// TIA Portal project "14_Palletizer_System" (V19)

(* hardware
DEVICE "S7-1500/ET200MP station_1"  S7-1500 station
   slot 0: "Rail_0"  Rack  6ES7 590-1***0-0AA0
   slot 1: "PLC_1"  CPU 1513-1 PN  6ES7 513-1AL02-0AB0  V2.9
      slot 3: "CPU display_1"  6ES7591-1AA00-0AA0
      slot 32768: "PROFINET interface_1"  X1
         slot 32769: "Port_1"  X1 P1
         slot 32770: "Port_2"  X1 P2
      slot 34817: "Virtual CP interface port_1"  Virtual CP interface port  Virtual CP interface port
*)

// ===== PLC "PLC_1"  CPU 1513-1 PN =====

VAR_GLOBAL   // PLC tag table "Default tag table"
   "Start" AT %I0.0 : Bool;
   "Stop" AT %I0.1 : Bool;
   "Reset" AT %I0.2 : Bool;
   "Auto" AT %I0.3 : Bool;
   "Manual" AT %I0.4 : Bool;
   "Box at entry" AT %I0.5 : Bool;
   "Clamped" AT %I0.6 : Bool;
   "Elevator moving" AT %I0.7 : Bool;
   "Pallet at entry" AT %I1.0 : Bool;
   "Pallet at exit" AT %I1.1 : Bool;
   "Pallet loaded" AT %I1.2 : Bool;
   "Plate limit" AT %I1.3 : Bool;
   "Pusher limit" AT %I1.4 : Bool;
   "Start light" AT %Q0.0 : Bool;
   "Stop light" AT %Q0.1 : Bool;
   "Reset light" AT %Q0.2 : Bool;
   "Clamp" AT %Q0.3 : Bool;
   "Box feeder" AT %Q0.4 : Bool;
   "Elevator up" AT %Q0.5 : Bool;
   "Elevator down" AT %Q0.6 : Bool;
   "Exit conveyor" AT %Q0.7 : Bool;
   "Load belt" AT %Q1.0 : Bool;
   "Load pallet" AT %Q1.1 : Bool;
   "Move to limit" AT %Q1.2 : Bool;
   "Open plate" AT %Q1.3 : Bool;
   "Pallet feeder" AT %Q1.4 : Bool;
   "Push" AT %Q1.5 : Bool;
   "Turn" AT %Q1.6 : Bool;
   "Warning light" AT %Q1.7 : Bool;
   "Set the value for the set of boxes" AT %ID30 : Real;
   "Counter" AT %QD30 : DInt;
   "Display for the set of box" AT %QD34 : DInt;
   "nw2" AT %M0.0 : Bool;
   "nw3 2nd memory" AT %M0.2 : Bool;
   "nw3 1st memory (Unpause)" AT %M0.1 : Bool;
   "nw4 pl p" AT %M1.1 : Bool;
   "nw4" AT %M0.3 : Bool;
   "nw4 op n" AT %M3.6 : Bool;
   "nw4 bae p" AT %M1.4 : Bool;
   "nw5" AT %M0.4 : Bool;
   "nw5 pl p" AT %M1.0 : Bool;
   "nw5 op n" AT %M3.7 : Bool;
   "nw6 bae n" AT %M1.2 : Bool;
   "nw6 bae p" AT %M1.3 : Bool;
   "nw6" AT %M4.0 : Bool;
   "nw6 pl p reset DB1" AT %M0.7 : Bool;
   "nw6 pl p" AT %M4.1 : Bool;
   "nw7 pae p" AT %M5.7 : Bool;
   "nw7" AT %M1.6 : Bool;
   "nw7 pl p" AT %M6.3 : Bool;
   "nw8 pae n" AT %M6.4 : Bool;
   "O/P for DB4 nw15" AT %M5.4 : Bool;
   "nw8" AT %M1.7 : Bool;
   "nw8 em n" AT %M6.0 : Bool;
   "nw8 pl p" AT %M2.6 : Bool;
   "nw9 pl p" AT %M2.4 : Bool;
   "nw9" AT %M2.0 : Bool;
   "nw9 em n" AT %M2.2 : Bool;
   "nw10 pl p" AT %M6.2 : Bool;
   "nw10" AT %M2.1 : Bool;
   "nw10 em n" AT %M2.3 : Bool;
   "nw10 pae p" AT %M6.1 : Bool;
   "nw11 p n" AT %M2.5 : Bool;
   "nw11" AT %M4.5 : Bool;
   "nw11 ed p reset CTU" AT %M3.5 : Bool;
   "nw11 ed p reset SR" AT %M4.6 : Bool;
   "nw13 pl p" AT %M3.1 : Bool;
   "nw13" AT %M3.4 : Bool;
   "nw12 c n" AT %M3.0 : Bool;
   "nw12" AT %M2.7 : Bool;
   "nw12 em n" AT %M3.2 : Bool;
   "nw13 pae p" AT %M5.6 : Bool;
   "nw14 p n" AT %M0.5 : Bool;
   "nw14 op n" AT %M4.4 : Bool;
   "nw14" AT %M4.2 : Bool;
   "nw14 ed p reset CTU" AT %M0.6 : Bool;
   "nw14 c n reset SR" AT %M4.3 : Bool;
   "nw15 ed n" AT %M4.7 : Bool;
   "nw15 pae p" AT %M5.0 : Bool;
   "Set the value for boxes on the display" AT %MW100 : Int;
   "nw16 pae n" AT %M5.1 : Bool;
   "nw16" AT %M5.3 : Bool;
   "nw16 eu p" AT %M6.7 : Bool;
   "nw17 bae n" AT %M6.5 : Bool;
   "nw18" AT %M6.6 : Bool;
   "nw13 op n" AT %M3.3 : Bool;
END_VAR

// folder: System blocks/Program resources

DATA_BLOCK "IEC_Counter_0_DB"   // DB1
{ S7_Optimized_Access := 'TRUE' }
AUTHOR : Simatic
FAMILY : IEC
NAME : CNTR
VERSION : 1.0
// stored: InstanceOfName IEC_COUNTER
"IEC_COUNTER"
BEGIN
END_DATA_BLOCK

DATA_BLOCK "IEC_Counter_0_DB_1"   // DB2
{ S7_Optimized_Access := 'TRUE' }
AUTHOR : Simatic
FAMILY : IEC
NAME : CNTR
VERSION : 1.0
// stored: InstanceOfName IEC_COUNTER
"IEC_COUNTER"
BEGIN
END_DATA_BLOCK

DATA_BLOCK "CTU to turn the box"   // DB3
{ S7_Optimized_Access := 'TRUE' }
AUTHOR : Simatic
FAMILY : IEC
NAME : CNTR
VERSION : 1.0
// stored: InstanceOfName IEC_COUNTER
"IEC_COUNTER"
BEGIN
END_DATA_BLOCK

DATA_BLOCK "Count a set of boxes that are moved on the pallet"   // DB4
{ S7_Optimized_Access := 'TRUE' }
AUTHOR : Simatic
FAMILY : IEC
NAME : CNTR
VERSION : 1.0
// stored: InstanceOfName IEC_COUNTER
"IEC_COUNTER"
BEGIN
END_DATA_BLOCK

DATA_BLOCK "Count total number of boxes that are moved on the pallet"   // DB5
{ S7_Optimized_Access := 'TRUE' }
AUTHOR : Simatic
FAMILY : IEC
NAME : CNTR
VERSION : 1.0
// stored: InstanceOfName IEC_COUNTER
"IEC_COUNTER"
BEGIN
END_DATA_BLOCK

// folder: (top level)

ORGANIZATION_BLOCK "Main"   // OB1, LAD, ProgramCycle
TITLE = "Main Program Sweep (Cycle)"
{ S7_Optimized_Access := 'TRUE' }
VERSION : 0.1
   VAR_INPUT
      Initial_Call : Bool;   // Initial call of this OB
      Remanence : Bool;   // =True, if remanent data are available
   END_VAR
   VAR_TEMP   // added for the SCL form of the ladder/FBD networks
      _w1 : Bool;
      _w2 : Bool;
      _w3 : Bool;
      _w4 : Bool;
   END_VAR
BEGIN

REGION Network 2: Start or Reset System with LED ON/OFF which are mounted on the switches
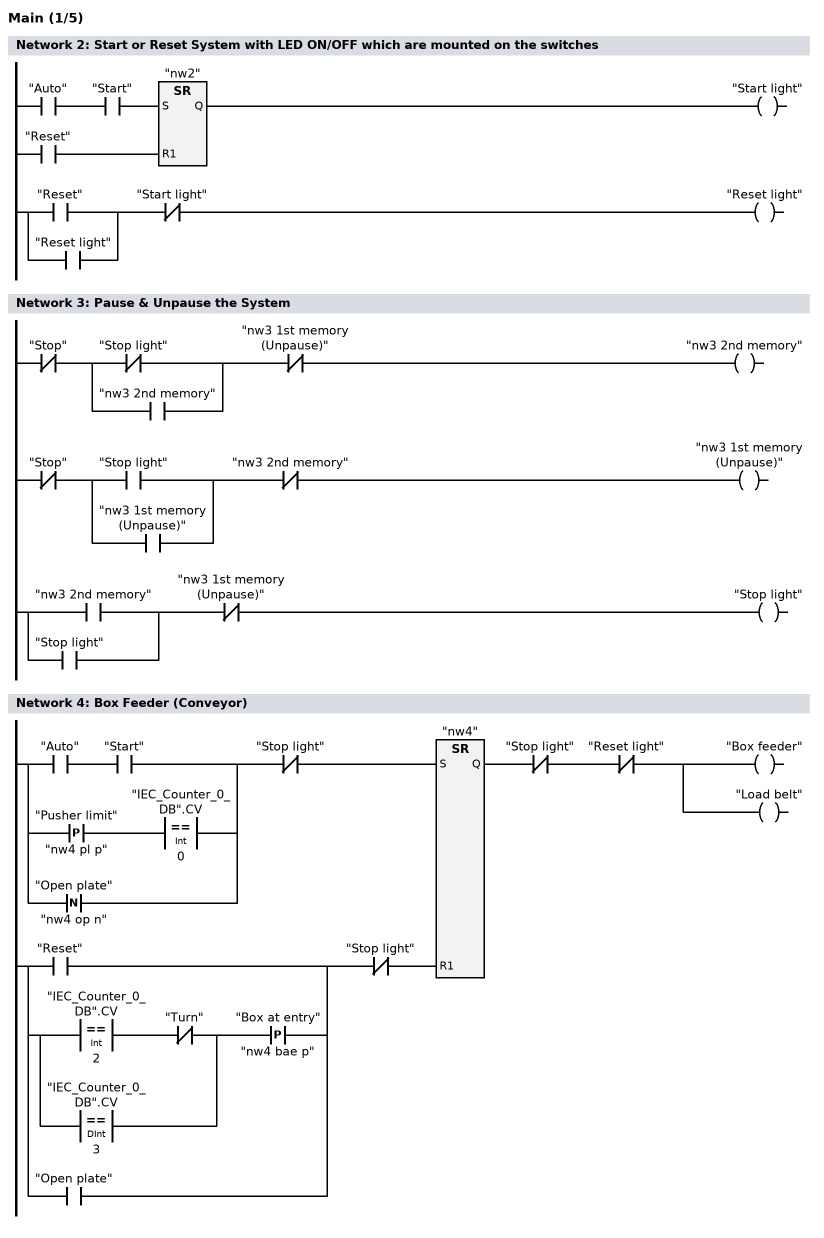
   RUNG wire#powerrail
      Contact( "Auto" )
      Contact( "Start" )
      S_SR(operand := "nw2", r1 := wire#w1)
      Coil( "Start light" )
   END_RUNG
   RUNG wire#powerrail
      Contact( "Reset" )
   END_RUNG wire#w1
   RUNG wire#powerrail
      Contact( "Reset" )
      wire#w2
      I_Contact( "Start light" )
      Coil( "Reset light" )
   END_RUNG
   RUNG wire#powerrail
      Contact( "Reset light" )
   END_RUNG wire#w2
   // the same network as SCL:
   IF "Auto" AND "Start" THEN
       "nw2" := TRUE;   // SR flip-flop
   END_IF;
   IF "Reset" THEN "nw2" := FALSE; END_IF;
   "Start light" := "nw2";
   "Reset light" := ("Reset" OR "Reset light") AND NOT "Start light";
END_REGION

REGION Network 3: Pause & Unpause the System
   RUNG wire#powerrail
      I_Contact( "Stop" )
      wire#w1
      I_Contact( "Stop light" )
      wire#w2
      I_Contact( "nw3 1st memory (Unpause)" )
      Coil( "nw3 2nd memory" )
   END_RUNG
   RUNG wire#w1
      Contact( "nw3 2nd memory" )
   END_RUNG wire#w2
   RUNG wire#powerrail
      I_Contact( "Stop" )
      wire#w3
      Contact( "Stop light" )
      wire#w4
      I_Contact( "nw3 2nd memory" )
      Coil( "nw3 1st memory (Unpause)" )
   END_RUNG
   RUNG wire#w3
      Contact( "nw3 1st memory (Unpause)" )
   END_RUNG wire#w4
   RUNG wire#powerrail
      Contact( "nw3 2nd memory" )
      wire#w5
      I_Contact( "nw3 1st memory (Unpause)" )
      Coil( "Stop light" )
   END_RUNG
   RUNG wire#powerrail
      Contact( "Stop light" )
   END_RUNG wire#w5
   // the same network as SCL:
   "nw3 2nd memory" := NOT "Stop" AND (NOT "Stop light" OR "nw3 2nd memory") AND NOT "nw3 1st memory (Unpause)";
   "nw3 1st memory (Unpause)" := NOT "Stop" AND ("Stop light" OR "nw3 1st memory (Unpause)") AND NOT "nw3 2nd memory";
   "Stop light" := ("nw3 2nd memory" OR "Stop light") AND NOT "nw3 1st memory (Unpause)";
END_REGION

REGION Network 4: Box Feeder (Conveyor)
   RUNG wire#powerrail
      Contact( "Auto" )
      Contact( "Start" )
      wire#w1
      I_Contact( "Stop light" )
      S_SR(operand := "nw4", r1 := wire#w4)
      I_Contact( "Stop light" )
      I_Contact( "Reset light" )
      wire#w5
      Coil( "Box feeder" )
   END_RUNG
   RUNG wire#powerrail
      P_Contact(operand := "Pusher limit", bit := "nw4 pl p")
      { S7_Templates := "SrcType := Int" } EQ_Contact(in1 := "IEC_Counter_0_DB".CV, in2 := 0)
   END_RUNG wire#w1
   RUNG wire#powerrail
      N_Contact(operand := "Open plate", bit := "nw4 op n")
   END_RUNG wire#w1
   RUNG wire#powerrail
      Contact( "Reset" )
      wire#w2
      I_Contact( "Stop light" )
   END_RUNG wire#w4
   RUNG wire#powerrail
      { S7_Templates := "SrcType := Int" } EQ_Contact(in1 := "IEC_Counter_0_DB".CV, in2 := 2)
      I_Contact( "Turn" )
      wire#w3
      P_Contact(operand := "Box at entry", bit := "nw4 bae p")
   END_RUNG wire#w2
   RUNG wire#powerrail
      { S7_Templates := "SrcType := DInt" } EQ_Contact(in1 := "IEC_Counter_0_DB".CV, in2 := 3)
   END_RUNG wire#w3
   RUNG wire#powerrail
      Contact( "Open plate" )
   END_RUNG wire#w2
   RUNG wire#w5
      Coil( "Load belt" )
   END_RUNG
   // the same network as SCL:
   #_w1 := "Pusher limit" AND NOT "nw4 pl p";   // rising edge of "Pusher limit"
   "nw4 pl p" := "Pusher limit";
   #_w2 := NOT "Open plate" AND "nw4 op n";   // falling edge of "Open plate"
   "nw4 op n" := "Open plate";
   #_w3 := ((("IEC_Counter_0_DB".CV = 2) AND NOT "Turn") OR ("IEC_Counter_0_DB".CV = 3)) AND "Box at entry" AND NOT "nw4 bae p";   // rising edge of "Box at entry"
   "nw4 bae p" := "Box at entry";
   IF (("Auto" AND "Start") OR (#_w1 AND ("IEC_Counter_0_DB".CV = 0)) OR #_w2) AND NOT "Stop light" THEN
       "nw4" := TRUE;   // SR flip-flop
   END_IF;
   IF ("Reset" OR #_w3 OR "Open plate") AND NOT "Stop light" THEN "nw4" := FALSE; END_IF;
   "Box feeder" := "nw4" AND NOT "Stop light" AND NOT "Reset light";
   "Load belt" := "Box feeder";
END_REGION

REGION Network 5: Load Belt Conveyor (Move to Network 4 for Optimizer)
END_REGION

REGION Network 6: Push and Push Limit
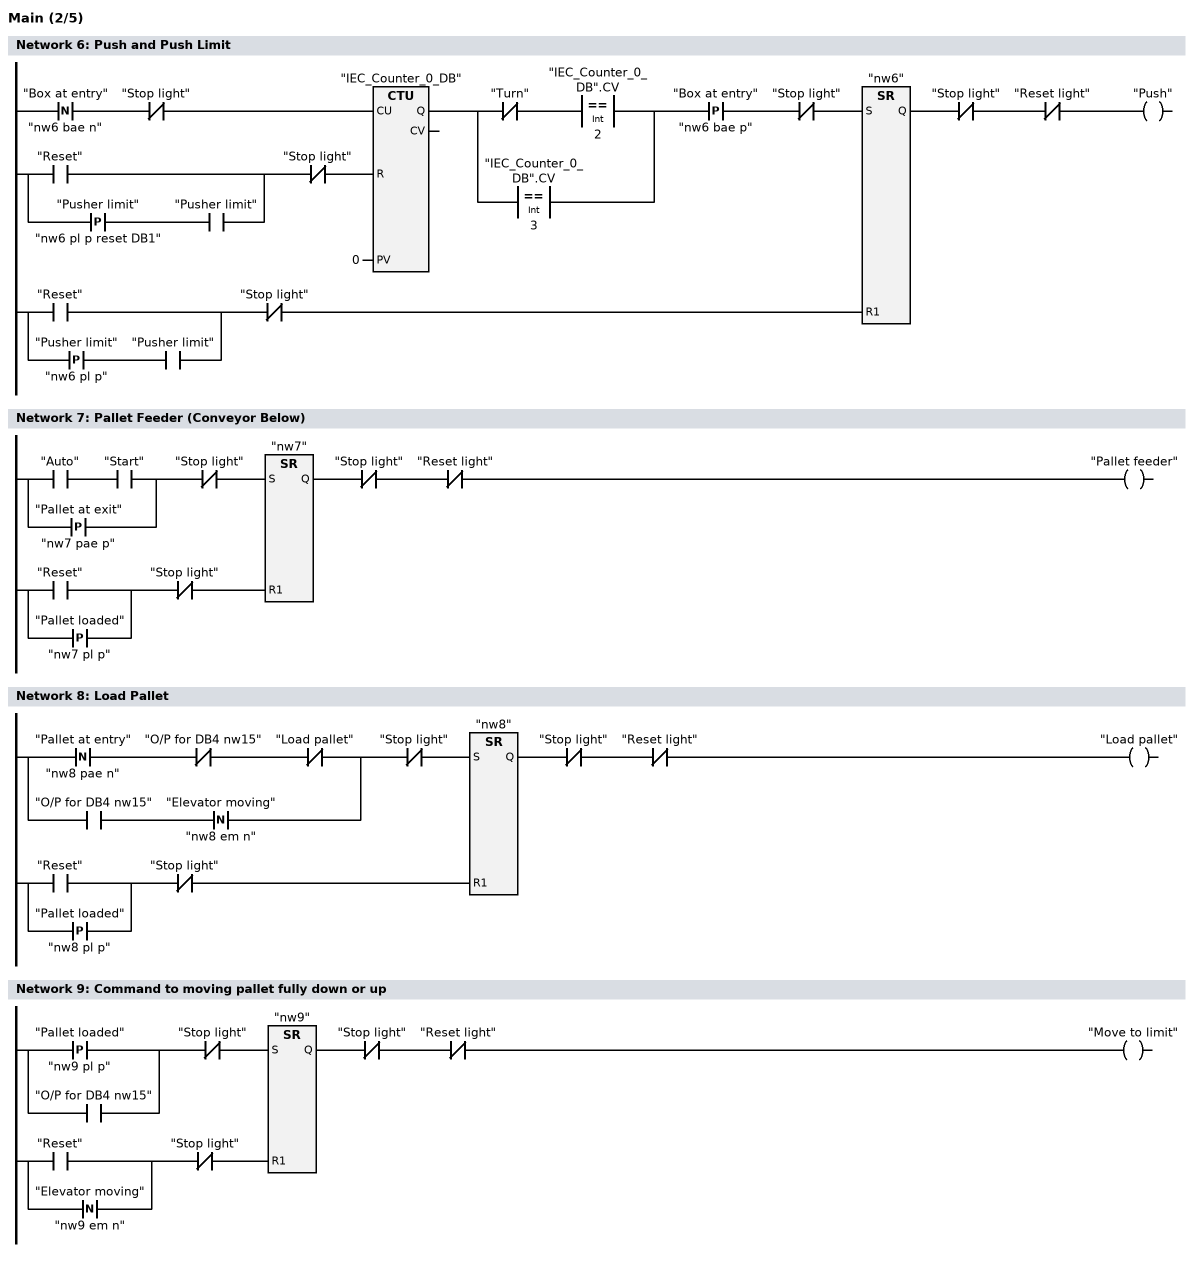
   #_w1 := NOT "Box at entry" AND "nw6 bae n";   // falling edge of "Box at entry"
   "nw6 bae n" := "Box at entry";
   #_w2 := "Pusher limit" AND NOT "nw6 pl p reset DB1";   // rising edge of "Pusher limit"
   "nw6 pl p reset DB1" := "Pusher limit";
   "IEC_Counter_0_DB".CTU(CU := #_w1 AND NOT "Stop light",
                          R := ("Reset" OR (#_w2 AND "Pusher limit")) AND NOT "Stop light",
                          PV := 0);
   #_w3 := "IEC_Counter_0_DB".Q AND ((NOT "Turn" AND ("IEC_Counter_0_DB".CV = 2)) OR ("IEC_Counter_0_DB".CV = 3)) AND "Box at entry" AND NOT "nw6 bae p";   // rising edge of "Box at entry"
   "nw6 bae p" := "Box at entry";
   #_w4 := "Pusher limit" AND NOT "nw6 pl p";   // rising edge of "Pusher limit"
   "nw6 pl p" := "Pusher limit";
   IF #_w3 AND NOT "Stop light" THEN
       "nw6" := TRUE;   // SR flip-flop
   END_IF;
   IF ("Reset" OR (#_w4 AND "Pusher limit")) AND NOT "Stop light" THEN "nw6" := FALSE; END_IF;
   "Push" := "nw6" AND NOT "Stop light" AND NOT "Reset light";
END_REGION

REGION Network 7: Pallet Feeder (Conveyor Below)
   RUNG wire#powerrail
      Contact( "Auto" )
      Contact( "Start" )
      wire#w1
      I_Contact( "Stop light" )
      S_SR(operand := "nw7", r1 := wire#w3)
      I_Contact( "Stop light" )
      I_Contact( "Reset light" )
      Coil( "Pallet feeder" )
   END_RUNG
   RUNG wire#powerrail
      P_Contact(operand := "Pallet at exit", bit := "nw7 pae p")
   END_RUNG wire#w1
   RUNG wire#powerrail
      Contact( "Reset" )
      wire#w2
      I_Contact( "Stop light" )
   END_RUNG wire#w3
   RUNG wire#powerrail
      P_Contact(operand := "Pallet loaded", bit := "nw7 pl p")
   END_RUNG wire#w2
   // the same network as SCL:
   #_w1 := "Pallet at exit" AND NOT "nw7 pae p";   // rising edge of "Pallet at exit"
   "nw7 pae p" := "Pallet at exit";
   #_w2 := "Pallet loaded" AND NOT "nw7 pl p";   // rising edge of "Pallet loaded"
   "nw7 pl p" := "Pallet loaded";
   IF (("Auto" AND "Start") OR #_w1) AND NOT "Stop light" THEN
       "nw7" := TRUE;   // SR flip-flop
   END_IF;
   IF ("Reset" OR #_w2) AND NOT "Stop light" THEN "nw7" := FALSE; END_IF;
   "Pallet feeder" := "nw7" AND NOT "Stop light" AND NOT "Reset light";
END_REGION

REGION Network 8: Load Pallet
   RUNG wire#powerrail
      N_Contact(operand := "Pallet at entry", bit := "nw8 pae n")
      I_Contact( "O/P for DB4 nw15" )
      I_Contact( "Load pallet" )
      wire#w1
      I_Contact( "Stop light" )
      S_SR(operand := "nw8", r1 := wire#w3)
      I_Contact( "Stop light" )
      I_Contact( "Reset light" )
      Coil( "Load pallet" )
   END_RUNG
   RUNG wire#powerrail
      Contact( "O/P for DB4 nw15" )
      N_Contact(operand := "Elevator moving", bit := "nw8 em n")
   END_RUNG wire#w1
   RUNG wire#powerrail
      Contact( "Reset" )
      wire#w2
      I_Contact( "Stop light" )
   END_RUNG wire#w3
   RUNG wire#powerrail
      P_Contact(operand := "Pallet loaded", bit := "nw8 pl p")
   END_RUNG wire#w2
   // the same network as SCL:
   #_w1 := NOT "Pallet at entry" AND "nw8 pae n";   // falling edge of "Pallet at entry"
   "nw8 pae n" := "Pallet at entry";
   #_w2 := "O/P for DB4 nw15" AND NOT "Elevator moving" AND "nw8 em n";   // falling edge of "Elevator moving"
   "nw8 em n" := "Elevator moving";
   #_w3 := "Pallet loaded" AND NOT "nw8 pl p";   // rising edge of "Pallet loaded"
   "nw8 pl p" := "Pallet loaded";
   IF ((#_w1 AND NOT "O/P for DB4 nw15" AND NOT "Load pallet") OR #_w2) AND NOT "Stop light" THEN
       "nw8" := TRUE;   // SR flip-flop
   END_IF;
   IF ("Reset" OR #_w3) AND NOT "Stop light" THEN "nw8" := FALSE; END_IF;
   "Load pallet" := "nw8" AND NOT "Stop light" AND NOT "Reset light";
END_REGION

REGION Network 9: Command to moving pallet fully down or up
   RUNG wire#powerrail
      P_Contact(operand := "Pallet loaded", bit := "nw9 pl p")
      wire#w1
      I_Contact( "Stop light" )
      S_SR(operand := "nw9", r1 := wire#w3)
      I_Contact( "Stop light" )
      I_Contact( "Reset light" )
      Coil( "Move to limit" )
   END_RUNG
   RUNG wire#powerrail
      Contact( "O/P for DB4 nw15" )
   END_RUNG wire#w1
   RUNG wire#powerrail
      Contact( "Reset" )
      wire#w2
      I_Contact( "Stop light" )
   END_RUNG wire#w3
   RUNG wire#powerrail
      N_Contact(operand := "Elevator moving", bit := "nw9 em n")
   END_RUNG wire#w2
   // the same network as SCL:
   #_w1 := "Pallet loaded" AND NOT "nw9 pl p";   // rising edge of "Pallet loaded"
   "nw9 pl p" := "Pallet loaded";
   #_w2 := NOT "Elevator moving" AND "nw9 em n";   // falling edge of "Elevator moving"
   "nw9 em n" := "Elevator moving";
   IF (#_w1 OR "O/P for DB4 nw15") AND NOT "Stop light" THEN
       "nw9" := TRUE;   // SR flip-flop
   END_IF;
   IF ("Reset" OR #_w2) AND NOT "Stop light" THEN "nw9" := FALSE; END_IF;
   "Move to limit" := "nw9" AND NOT "Stop light" AND NOT "Reset light";
END_REGION

REGION Network 10: Move Pallet upward by 1 step or fully up
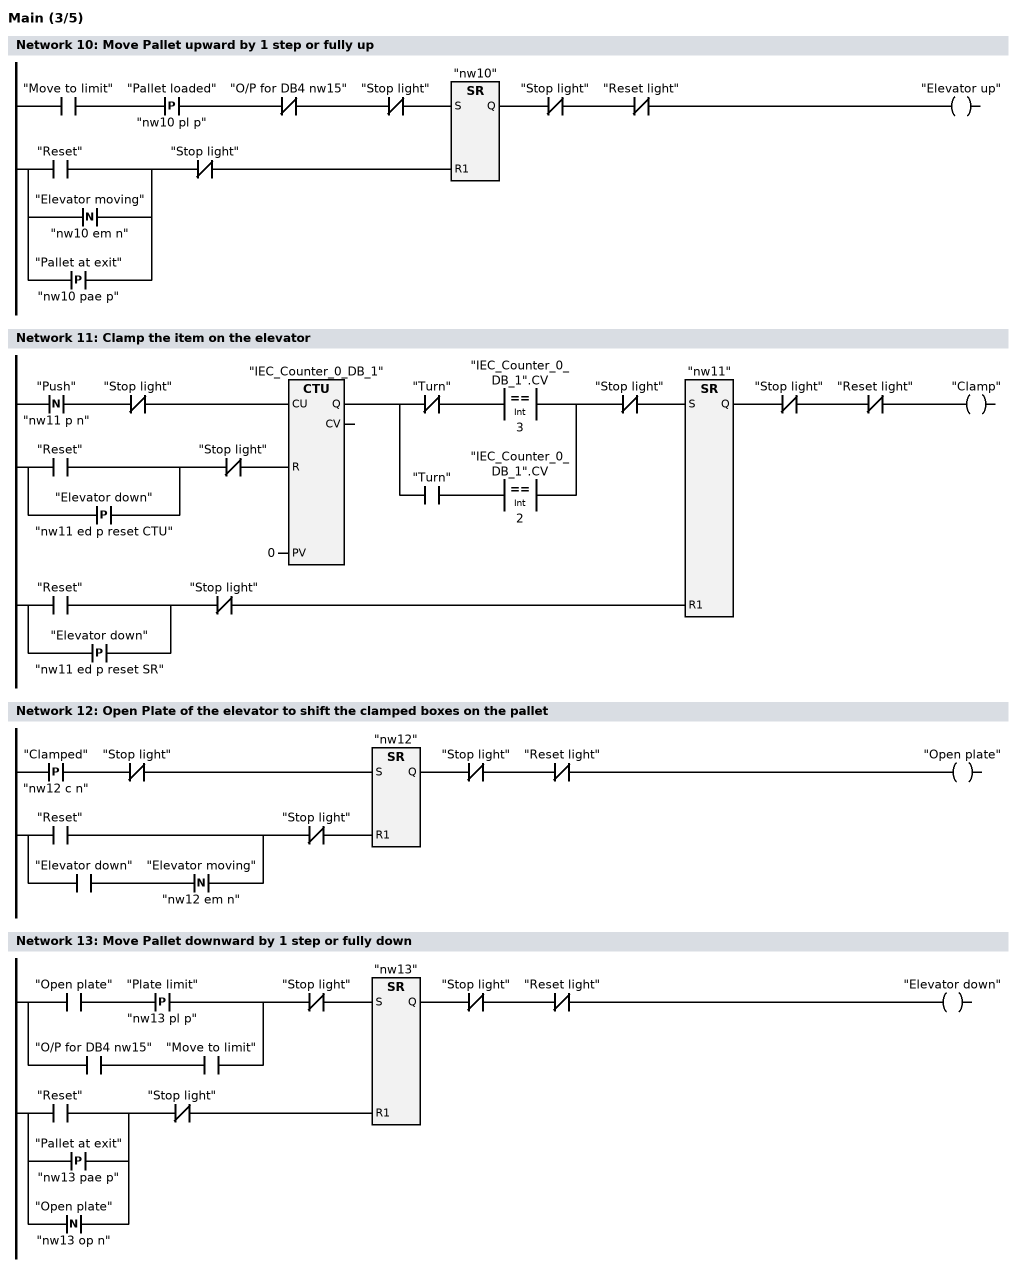
   RUNG wire#powerrail
      Contact( "Move to limit" )
      P_Contact(operand := "Pallet loaded", bit := "nw10 pl p")
      I_Contact( "O/P for DB4 nw15" )
      I_Contact( "Stop light" )
      S_SR(operand := "nw10", r1 := wire#w2)
      I_Contact( "Stop light" )
      I_Contact( "Reset light" )
      Coil( "Elevator up" )
   END_RUNG
   RUNG wire#powerrail
      Contact( "Reset" )
      wire#w1
      I_Contact( "Stop light" )
   END_RUNG wire#w2
   RUNG wire#powerrail
      N_Contact(operand := "Elevator moving", bit := "nw10 em n")
   END_RUNG wire#w1
   RUNG wire#powerrail
      P_Contact(operand := "Pallet at exit", bit := "nw10 pae p")
   END_RUNG wire#w1
   // the same network as SCL:
   #_w1 := "Move to limit" AND "Pallet loaded" AND NOT "nw10 pl p";   // rising edge of "Pallet loaded"
   "nw10 pl p" := "Pallet loaded";
   #_w2 := NOT "Elevator moving" AND "nw10 em n";   // falling edge of "Elevator moving"
   "nw10 em n" := "Elevator moving";
   #_w3 := "Pallet at exit" AND NOT "nw10 pae p";   // rising edge of "Pallet at exit"
   "nw10 pae p" := "Pallet at exit";
   IF #_w1 AND NOT "O/P for DB4 nw15" AND NOT "Stop light" THEN
       "nw10" := TRUE;   // SR flip-flop
   END_IF;
   IF ("Reset" OR #_w2 OR #_w3) AND NOT "Stop light" THEN "nw10" := FALSE; END_IF;
   "Elevator up" := "nw10" AND NOT "Stop light" AND NOT "Reset light";
END_REGION

REGION Network 11: Clamp the item on the elevator
   #_w1 := NOT "Push" AND "nw11 p n";   // falling edge of "Push"
   "nw11 p n" := "Push";
   #_w2 := "Elevator down" AND NOT "nw11 ed p reset CTU";   // rising edge of "Elevator down"
   "nw11 ed p reset CTU" := "Elevator down";
   "IEC_Counter_0_DB_1".CTU(CU := #_w1 AND NOT "Stop light",
                           R := ("Reset" OR #_w2) AND NOT "Stop light",
                           PV := 0);
   #_w3 := "Elevator down" AND NOT "nw11 ed p reset SR";   // rising edge of "Elevator down"
   "nw11 ed p reset SR" := "Elevator down";
   IF "IEC_Counter_0_DB_1".Q AND ((NOT "Turn" AND ("IEC_Counter_0_DB_1".CV = 3)) OR ("Turn" AND ("IEC_Counter_0_DB_1".CV = 2))) AND NOT "Stop light" THEN
       "nw11" := TRUE;   // SR flip-flop
   END_IF;
   IF ("Reset" OR #_w3) AND NOT "Stop light" THEN "nw11" := FALSE; END_IF;
   "Clamp" := "nw11" AND NOT "Stop light" AND NOT "Reset light";
END_REGION

REGION Network 12: Open Plate of the elevator to shift the clamped boxes on the pallet
   RUNG wire#powerrail
      P_Contact(operand := "Clamped", bit := "nw12 c n")
      I_Contact( "Stop light" )
      S_SR(operand := "nw12", r1 := wire#w2)
      I_Contact( "Stop light" )
      I_Contact( "Reset light" )
      Coil( "Open plate" )
   END_RUNG
   RUNG wire#powerrail
      Contact( "Reset" )
      wire#w1
      I_Contact( "Stop light" )
   END_RUNG wire#w2
   RUNG wire#powerrail
      Contact( "Elevator down" )
      N_Contact(operand := "Elevator moving", bit := "nw12 em n")
   END_RUNG wire#w1
   // the same network as SCL:
   #_w1 := "Clamped" AND NOT "nw12 c n";   // rising edge of "Clamped"
   "nw12 c n" := "Clamped";
   #_w2 := "Elevator down" AND NOT "Elevator moving" AND "nw12 em n";   // falling edge of "Elevator moving"
   "nw12 em n" := "Elevator moving";
   IF #_w1 AND NOT "Stop light" THEN
       "nw12" := TRUE;   // SR flip-flop
   END_IF;
   IF ("Reset" OR #_w2) AND NOT "Stop light" THEN "nw12" := FALSE; END_IF;
   "Open plate" := "nw12" AND NOT "Stop light" AND NOT "Reset light";
END_REGION

REGION Network 13: Move Pallet downward by 1 step or fully down
   RUNG wire#powerrail
      Contact( "Open plate" )
      P_Contact(operand := "Plate limit", bit := "nw13 pl p")
      wire#w1
      I_Contact( "Stop light" )
      S_SR(operand := "nw13", r1 := wire#w3)
      I_Contact( "Stop light" )
      I_Contact( "Reset light" )
      Coil( "Elevator down" )
   END_RUNG
   RUNG wire#powerrail
      Contact( "O/P for DB4 nw15" )
      Contact( "Move to limit" )
   END_RUNG wire#w1
   RUNG wire#powerrail
      Contact( "Reset" )
      wire#w2
      I_Contact( "Stop light" )
   END_RUNG wire#w3
   RUNG wire#powerrail
      P_Contact(operand := "Pallet at exit", bit := "nw13 pae p")
   END_RUNG wire#w2
   RUNG wire#powerrail
      N_Contact(operand := "Open plate", bit := "nw13 op n")
   END_RUNG wire#w2
   // the same network as SCL:
   #_w1 := "Open plate" AND "Plate limit" AND NOT "nw13 pl p";   // rising edge of "Plate limit"
   "nw13 pl p" := "Plate limit";
   #_w2 := "Pallet at exit" AND NOT "nw13 pae p";   // rising edge of "Pallet at exit"
   "nw13 pae p" := "Pallet at exit";
   #_w3 := NOT "Open plate" AND "nw13 op n";   // falling edge of "Open plate"
   "nw13 op n" := "Open plate";
   IF (#_w1 OR ("O/P for DB4 nw15" AND "Move to limit")) AND NOT "Stop light" THEN
       "nw13" := TRUE;   // SR flip-flop
   END_IF;
   IF ("Reset" OR #_w2 OR #_w3) AND NOT "Stop light" THEN "nw13" := FALSE; END_IF;
   "Elevator down" := "nw13" AND NOT "Stop light" AND NOT "Reset light";
END_REGION

REGION Network 14: Turn box 90 degree clockwise
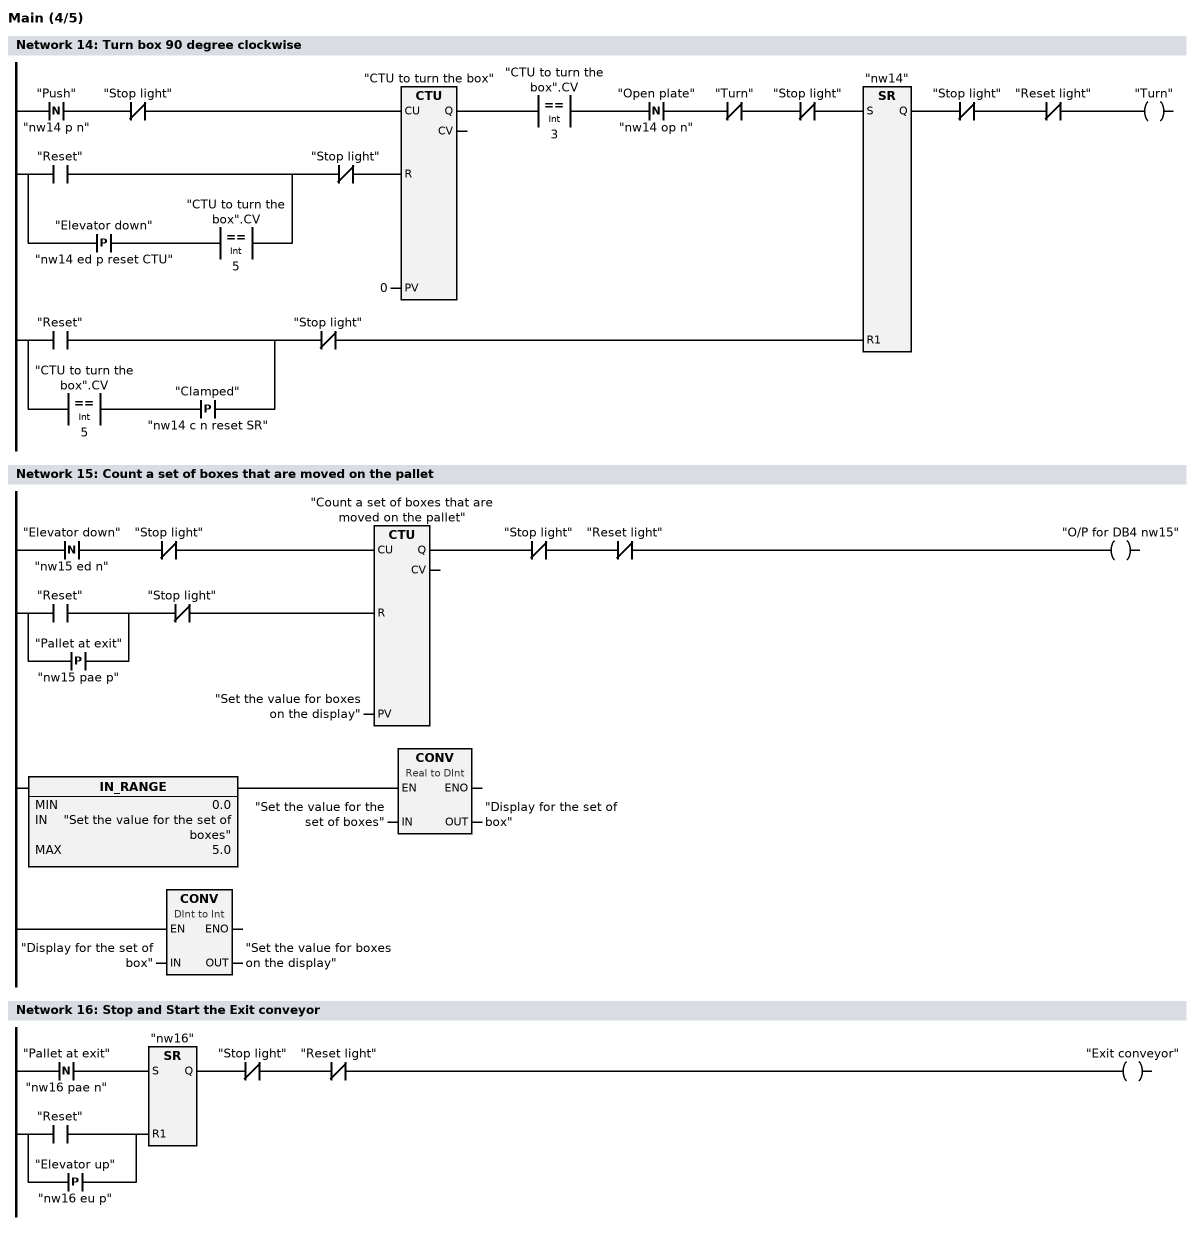
   #_w1 := NOT "Push" AND "nw14 p n";   // falling edge of "Push"
   "nw14 p n" := "Push";
   #_w2 := "Elevator down" AND NOT "nw14 ed p reset CTU";   // rising edge of "Elevator down"
   "nw14 ed p reset CTU" := "Elevator down";
   "CTU to turn the box".CTU(CU := #_w1 AND NOT "Stop light",
                           R := ("Reset" OR (#_w2 AND ("CTU to turn the box".CV = 5))) AND NOT "Stop light",
                           PV := 0);
   #_w3 := "CTU to turn the box".Q AND ("CTU to turn the box".CV = 3) AND NOT "Open plate" AND "nw14 op n";   // falling edge of "Open plate"
   "nw14 op n" := "Open plate";
   #_w4 := ("CTU to turn the box".CV = 5) AND "Clamped" AND NOT "nw14 c n reset SR";   // rising edge of "Clamped"
   "nw14 c n reset SR" := "Clamped";
   IF #_w3 AND NOT "Turn" AND NOT "Stop light" THEN
       "nw14" := TRUE;   // SR flip-flop
   END_IF;
   IF ("Reset" OR #_w4) AND NOT "Stop light" THEN "nw14" := FALSE; END_IF;
   "Turn" := "nw14" AND NOT "Stop light" AND NOT "Reset light";
END_REGION

REGION Network 15: Count a set of boxes that are moved on the pallet
   #_w1 := NOT "Elevator down" AND "nw15 ed n";   // falling edge of "Elevator down"
   "nw15 ed n" := "Elevator down";
   #_w2 := "Pallet at exit" AND NOT "nw15 pae p";   // rising edge of "Pallet at exit"
   "nw15 pae p" := "Pallet at exit";
   "Count a set of boxes that are moved on the pallet".CTU(CU := #_w1 AND NOT "Stop light",
                           R := ("Reset" OR #_w2) AND NOT "Stop light",
                           PV := "Set the value for boxes on the display");
   "O/P for DB4 nw15" := "Count a set of boxes that are moved on the pallet".Q AND NOT "Stop light" AND NOT "Reset light";
   IF (0.0 <= "Set the value for the set of boxes") AND ("Set the value for the set of boxes" <= 5.0) THEN
       "Display for the set of box" := REAL_TO_DINT("Set the value for the set of boxes");
   END_IF;
   "Set the value for boxes on the display" := DINT_TO_INT("Display for the set of box");
END_REGION

REGION Network 16: Stop and Start the Exit conveyor
   RUNG wire#powerrail
      N_Contact(operand := "Pallet at exit", bit := "nw16 pae n")
      S_SR(operand := "nw16", r1 := wire#w1)
      I_Contact( "Stop light" )
      I_Contact( "Reset light" )
      Coil( "Exit conveyor" )
   END_RUNG
   RUNG wire#powerrail
      Contact( "Reset" )
   END_RUNG wire#w1
   RUNG wire#powerrail
      P_Contact(operand := "Elevator up", bit := "nw16 eu p")
   END_RUNG wire#w1
   // the same network as SCL:
   #_w1 := NOT "Pallet at exit" AND "nw16 pae n";   // falling edge of "Pallet at exit"
   "nw16 pae n" := "Pallet at exit";
   #_w2 := "Elevator up" AND NOT "nw16 eu p";   // rising edge of "Elevator up"
   "nw16 eu p" := "Elevator up";
   IF #_w1 THEN
       "nw16" := TRUE;   // SR flip-flop
   END_IF;
   IF "Reset" OR #_w2 THEN "nw16" := FALSE; END_IF;
   "Exit conveyor" := "nw16" AND NOT "Stop light" AND NOT "Reset light";
END_REGION

REGION Network 17: Count the total number of boxes that are moved on the pallet
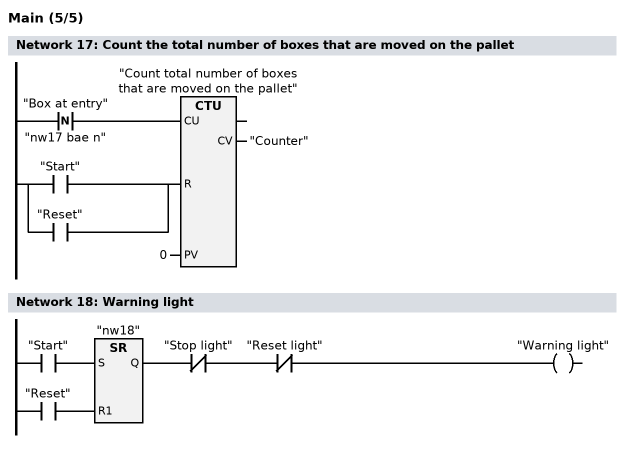
   #_w1 := NOT "Box at entry" AND "nw17 bae n";   // falling edge of "Box at entry"
   "nw17 bae n" := "Box at entry";
   "Count total number of boxes that are moved on the pallet".CTU(CU := #_w1,
                           R := "Start" OR "Reset",
                           PV := 0,
                           CV => "Counter");
END_REGION

REGION Network 18: Warning light
   RUNG wire#powerrail
      Contact( "Start" )
      S_SR(operand := "nw18", r1 := wire#w1)
      I_Contact( "Stop light" )
      I_Contact( "Reset light" )
      Coil( "Warning light" )
   END_RUNG
   RUNG wire#powerrail
      Contact( "Reset" )
   END_RUNG wire#w1
   // the same network as SCL:
   IF "Start" THEN
       "nw18" := TRUE;   // SR flip-flop
   END_IF;
   IF "Reset" THEN "nw18" := FALSE; END_IF;
   "Warning light" := "nw18" AND NOT "Stop light" AND NOT "Reset light";
END_REGION
END_ORGANIZATION_BLOCK